FUNCTION_BLOCK TcoSequenceTestChildState EXTENDS TcoCore.TcoState
VAR
	_requestedState : UINT;
	_requestedStateCount :ULINT;
	_restoreCount :ULINT;
END_VAR

(*~
	<docu>
		<summary>
			This method is called on each change of the <c>State</c>. This method could be overloaded and custom code should be placed here.	
		</summary>			
	</docu>	
~*)
METHOD PROTECTED OnStateChange
VAR_INPUT
	PreviousState	: INT;
	NewState 		: INT;
END_VAR
IF NewState =  _requestedState THEN
	_requestedStateCount := _requestedStateCount + 1;
END_IF

IF NewState =  -1 THEN
	_restoreCount := _restoreCount + 1;
END_IF
END_METHOD

PROPERTY RequestedState : UINT
GET
RequestedState := _requestedState;
END_GET
SET
_requestedState := RequestedState;
END_SET
END_PROPERTY

END_FUNCTION_BLOCK

(* stored: Version 1.1.0.1
   POU TcoSequenceTestChildState: Id {c732740a-c3d3-0a45-32ab-d6759ebf7cd7}, SpecialFunc None
   Method OnStateChange: Id {20cacacd-9b7f-0c6f-262e-75334e647cb0}
   Property RequestedState: Id {8a2c40dd-2aa8-0a57-0fcc-9ddd84998dd2}
   Get Get: Id {f91adf27-34dc-0f72-3ca8-ed0cd0348baa}
   Set Set: Id {5a58aa0d-76d7-048c-2aa2-6781afa3914b} *)
